// TIA Portal V17 export
// export: Created 2024-10-17T14:16:17.4257296Z, ExportSetting WithDefaults, DisplayName Totally Integrated Automation Portal, DisplayVersion V17 Update 4, DisplayName TIA Portal Openness, DisplayVersion V17 Update 4, DisplayName TIA Portal Version Control Interface, DisplayVersion V17, DisplayName SINAMICS Startdrive Advanced, DisplayVersion V17 Update2, DisplayName SINAMICS Startdrive G130, G150, S120, S150, SINAMICS MV, S210, DisplayVersion V17 Update2, DisplayName SINAMICS Startdrive G110M, G120, G120C, G120D, G120P, G115D, DisplayVersion V17 Update2, DisplayName STEP 7 Professional, DisplayVersion V17 Update 4, DisplayName STEP 7 Safety, DisplayVersion V17, DisplayName WinCC Advanced / Unified PC, DisplayVersion V17 Update 4
TYPE "LPMLV2022_typeCommandRecipe"
TITLE = LPMLV2022_typeCommandRecipe
// Support: tech.team.motioncontrol@siemens.com
// stored: IsFailsafeCompliant false
   STRUCT
      ID : DInt;   // ID Value of the Recipe. The ID is used to indicate to the machine which recipe is being produced
      "Name" : String[80];   // Name of Recipe. The Recipe Name is used to further identify the product being produced, especially when alphanumeric characters are used (i.e. SKU or UPC)
      Unit : String[6];   // Unit of Measure of Recipe. The Recipe Unit is used to describe the unit of production for the product being produced
      PrimaryQty : Real;   // Primary Quantity Value of Recipe. PrimaryQty is used to provide a common reference for manufacturing throughput across all the machines on a production line. This element describes the number of Primary Products per recipe Unit for the product being produced by this unit/machine
      ProcessVariables : "LPMLV2022_typeCommandProcessVariables";   // Process Variables for each Recipe. The ProcessVariables structure can be used to hold particular set points needed by the unit/machine for the processing of a specific recipe
      Ingredients : "LPMLV2022_typeCommandIngredients";   // Ingredient Information for each Recipe. The Ingredients structure can be used to hold information for the raw materials that are used by the unit/machine in the processing of a particular product or recipe
   END_STRUCT;
END_TYPE
